Xinje XDPPro project, PLC1: XDH-60T4 (software 3.7.18 2024-11-27)

PROGRAM 梯形图

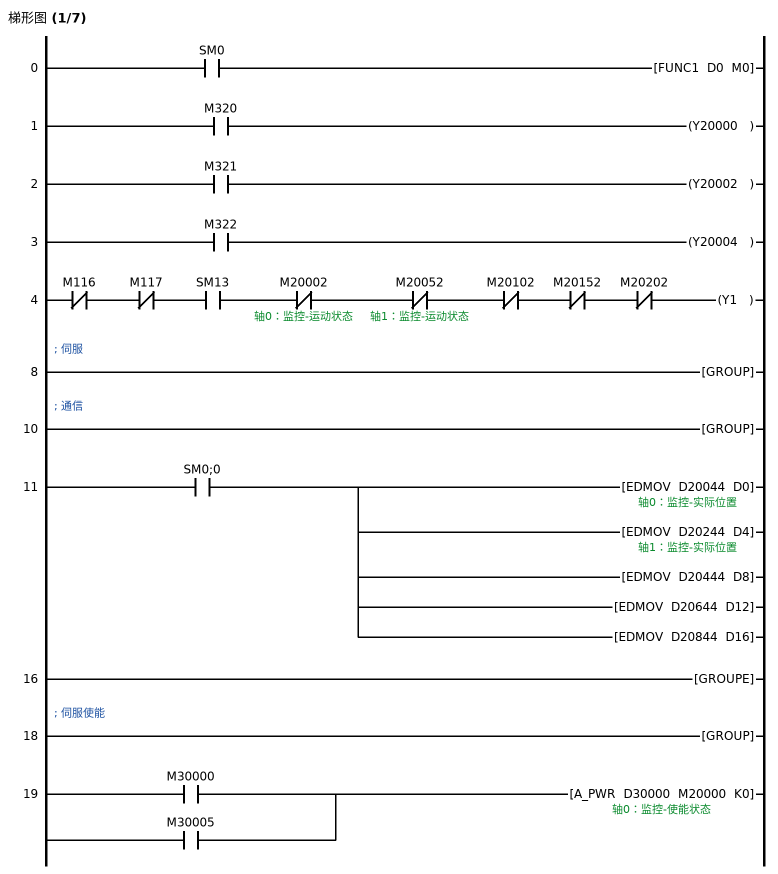
LD     SM0
FUNC1  D0 M0
LD     M320
OUT    Y20000
LD     M321
OUT    Y20002
LD     M322
OUT    Y20004
LDI    M116
ANI    M117
AND    SM13
ANI    M20002	; 轴0：监控-运动状态
ANI    M20052	; 轴1：监控-运动状态
ANI    M20102
ANI    M20152
ANI    M20202
OUT    Y1
; 伺服
GROUP
; 通信
GROUP
LD     SM0;0
EDMOV  D20044 D0	; 轴0：监控-实际位置
EDMOV  D20244 D4	; 轴1：监控-实际位置
EDMOV  D20444 D8
EDMOV  D20644 D12
EDMOV  D20844 D16
GROUPE
; 伺服使能
GROUP
LD     M30000
OR     M30005
A_PWR  D30000 M20000 K0	; 轴0：监控-使能状态

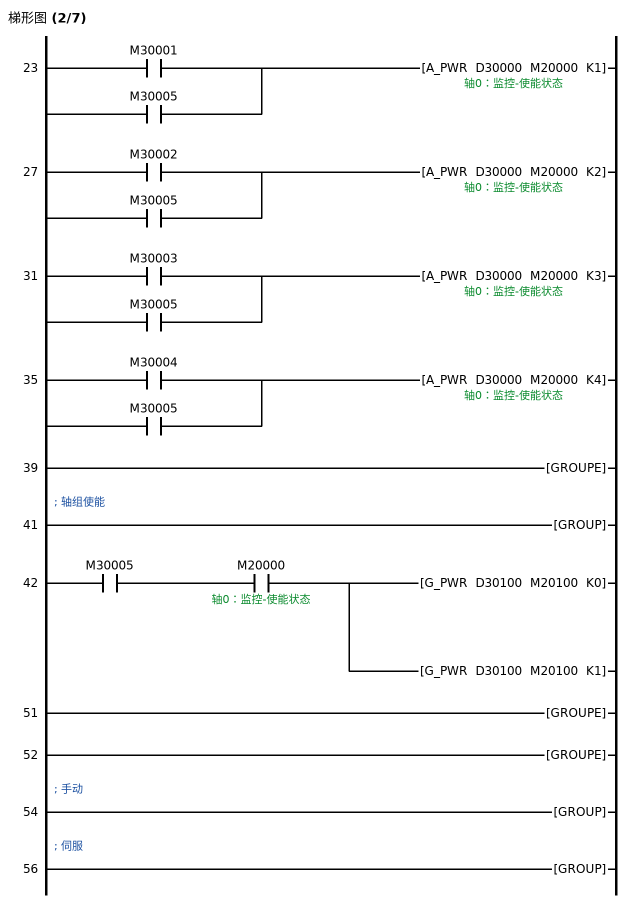
LD     M30001
OR     M30005
A_PWR  D30000 M20000 K1	; 轴0：监控-使能状态
LD     M30002
OR     M30005
A_PWR  D30000 M20000 K2	; 轴0：监控-使能状态
LD     M30003
OR     M30005
A_PWR  D30000 M20000 K3	; 轴0：监控-使能状态
LD     M30004
OR     M30005
A_PWR  D30000 M20000 K4	; 轴0：监控-使能状态
GROUPE
; 轴组使能
GROUP
LD     M30005
AND    M20000	; 轴0：监控-使能状态
G_PWR  D30100 M20100 K0
G_PWR  D30100 M20100 K1
GROUPE
GROUPE
; 手动
GROUP
; 伺服
GROUP

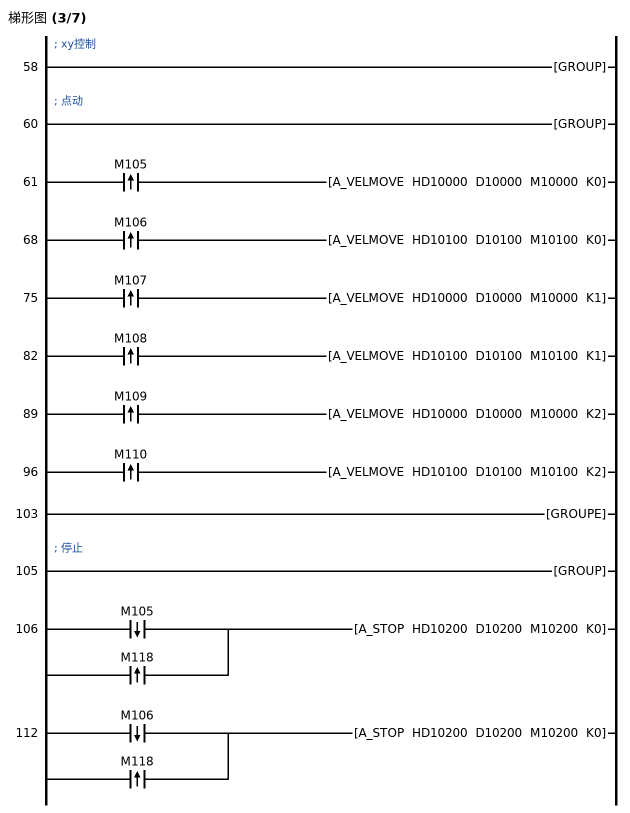
; xy控制
GROUP
; 点动
GROUP
LDP    M105
A_VELMOVE HD10000 D10000 M10000 K0
LDP    M106
A_VELMOVE HD10100 D10100 M10100 K0
LDP    M107
A_VELMOVE HD10000 D10000 M10000 K1
LDP    M108
A_VELMOVE HD10100 D10100 M10100 K1
LDP    M109
A_VELMOVE HD10000 D10000 M10000 K2
LDP    M110
A_VELMOVE HD10100 D10100 M10100 K2
GROUPE
; 停止
GROUP
LDF    M105
ORP    M118
A_STOP HD10200 D10200 M10200 K0
LDF    M106
ORP    M118
A_STOP HD10200 D10200 M10200 K0

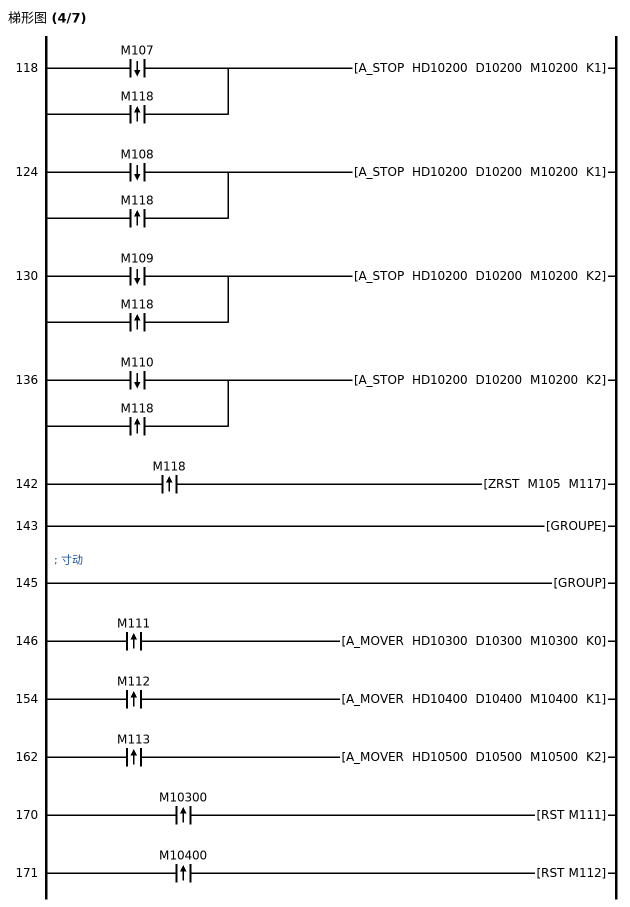
LDF    M107
ORP    M118
A_STOP HD10200 D10200 M10200 K1
LDF    M108
ORP    M118
A_STOP HD10200 D10200 M10200 K1
LDF    M109
ORP    M118
A_STOP HD10200 D10200 M10200 K2
LDF    M110
ORP    M118
A_STOP HD10200 D10200 M10200 K2
LDP    M118
ZRST   M105 M117
GROUPE
; 寸动
GROUP
LDP    M111
A_MOVER HD10300 D10300 M10300 K0
LDP    M112
A_MOVER HD10400 D10400 M10400 K1
LDP    M113
A_MOVER HD10500 D10500 M10500 K2
LDP    M10300
RST    M111
LDP    M10400
RST    M112

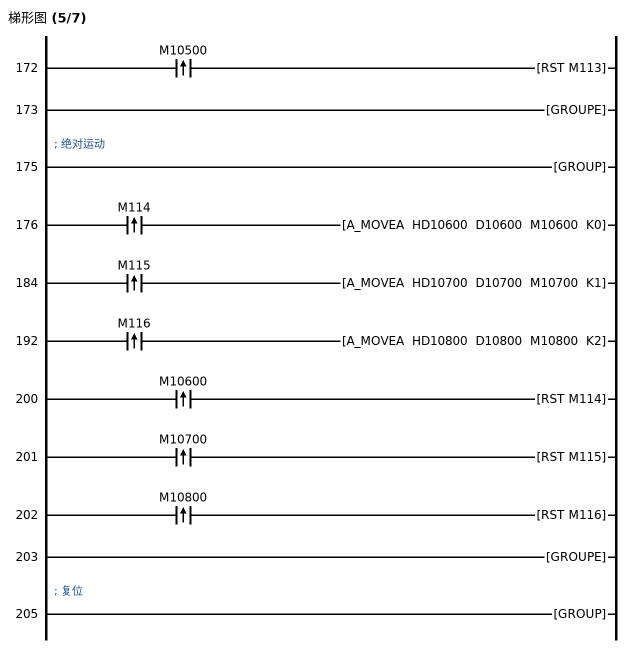
LDP    M10500
RST    M113
GROUPE
; 绝对运动
GROUP
LDP    M114
A_MOVEA HD10600 D10600 M10600 K0
LDP    M115
A_MOVEA HD10700 D10700 M10700 K1
LDP    M116
A_MOVEA HD10800 D10800 M10800 K2
LDP    M10600
RST    M114
LDP    M10700
RST    M115
LDP    M10800
RST    M116
GROUPE
; 复位
GROUP

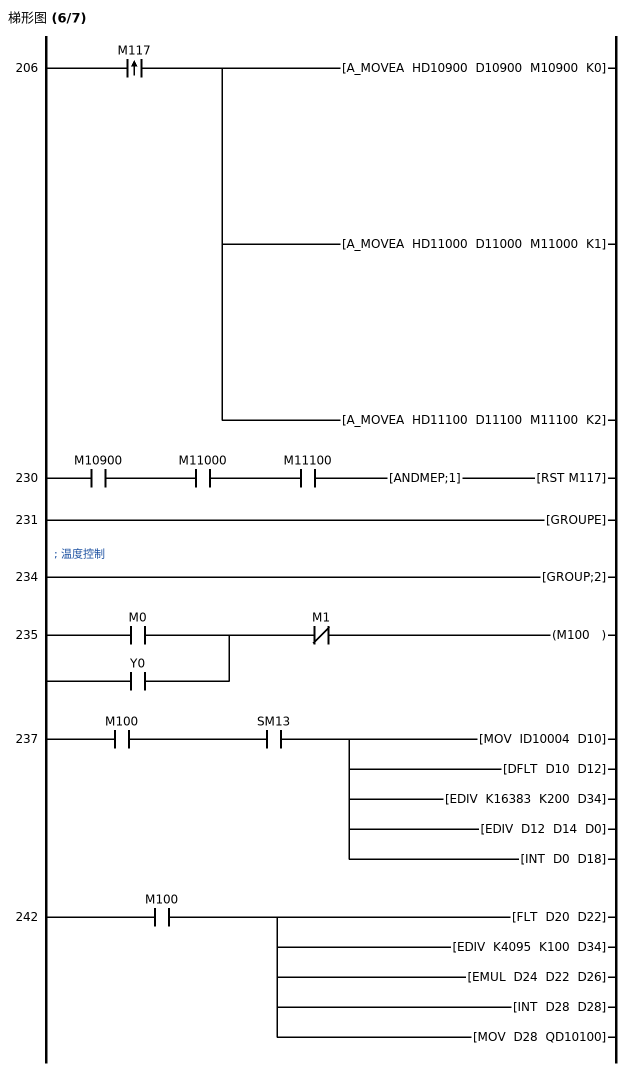
LDP    M117
A_MOVEA HD10900 D10900 M10900 K0
A_MOVEA HD11000 D11000 M11000 K1
A_MOVEA HD11100 D11100 M11100 K2
LD     M10900
AND    M11000
AND    M11100
ANDMEP;1
RST    M117
GROUPE
; 温度控制
GROUP;2
LD     M0
OR     Y0
ANI    M1
OUT    M100
LD     M100
AND    SM13
MOV    ID10004 D10
DFLT   D10 D12
EDIV   K16383 K200 D34
EDIV   D12 D14 D0
INT    D0 D18
LD     M100
FLT    D20 D22
EDIV   K4095 K100 D34
EMUL   D24 D22 D26
INT    D28 D28
MOV    D28 QD10100

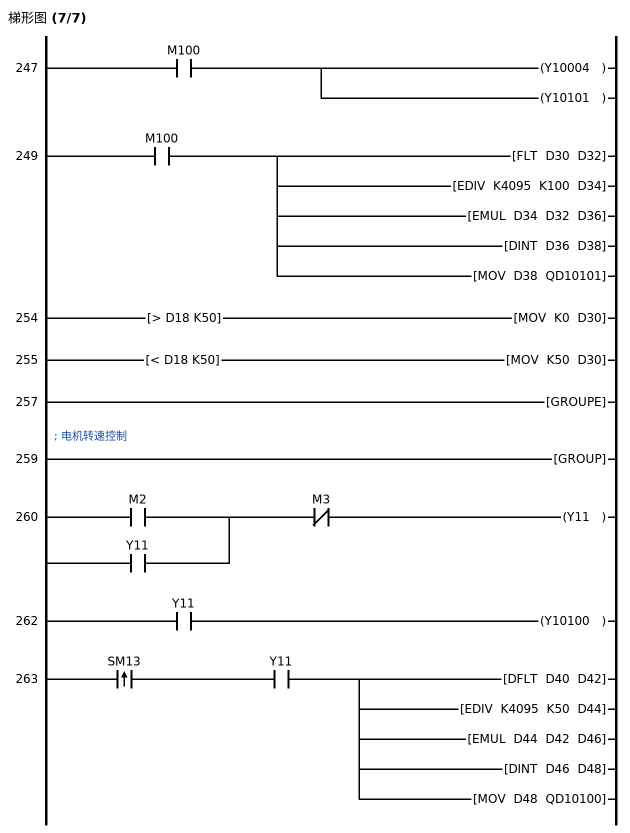
LD     M100
OUT    Y10004
OUT    Y10101
LD     M100
FLT    D30 D32
EDIV   K4095 K100 D34
EMUL   D34 D32 D36
DINT   D36 D38
MOV    D38 QD10101
LD>    D18 K50
MOV    K0 D30
LD<    D18 K50
MOV    K50 D30
GROUPE
; 电机转速控制
GROUP
LD     M2
OR     Y11
ANI    M3
OUT    Y11
LD     Y11
OUT    Y10100
LDP    SM13
AND    Y11
DFLT   D40 D42
EDIV   K4095 K50 D44
EMUL   D44 D42 D46
DINT   D46 D48
MOV    D48 QD10100

COMMENTS (devices not used above)
D20000	轴0：监控-状态机
D20200	轴1：监控-状态机
D20001	轴0：监控-错误码
D20201	轴1：监控-错误码
D20002	轴0：监控-调试模式
D20202	轴1：监控-调试模式
D20012	轴0：监控-目标位置
D20212	轴1：监控-目标位置
D20016	轴0：监控-指令位置
D20216	轴1：监控-指令位置
D20020	轴0：监控-指令速度
D20220	轴1：监控-指令速度
D20048	轴0：监控-实际速度
D20248	轴1：监控-实际速度
D20024	轴0：监控-实际加速度
D20224	轴1：监控-实际加速度
D20032	轴0：监控-指令转矩
D20232	轴1：监控-指令转矩
D20052	轴0：监控-实际转矩
D20252	轴1：监控-实际转矩
M20050	轴1：监控-使能状态
M20001	轴0：监控-错误状态
M20051	轴1：监控-错误状态
M20003	轴0：监控-定位状态
M20053	轴1：监控-定位状态
M20004	轴0：监控-原点开关
M20054	轴1：监控-原点开关
M20008	轴0：监控-指令完成状态
M20058	轴1：监控-指令完成状态
M20031	轴0：监控-正软限位
M20081	轴1：监控-正软限位
M20032	轴0：监控-负软限位
M20082	轴1：监控-负软限位
M20029	轴0：监控-正硬限位
M20079	轴1：监控-正硬限位
M20030	轴0：监控-负硬限位
M20080	轴1：监控-负硬限位
D20104	轴0：调试-启用轴调试
D20304	轴1：调试-启用轴调试
D20105	轴0：调试-运动类型
D20305	轴1：调试-运动类型
D20108	轴0：调试-目标位置
D20308	轴1：调试-目标位置
D20112	轴0：调试-速度
D20312	轴1：调试-速度
D20116	轴0：调试-加速度
D20316	轴1：调试-加速度
D20120	轴0：调试-减速度
D20320	轴1：调试-减速度
D20124	轴0：调试-加加速度
D20324	轴1：调试-加加速度
D20128	轴0：调试-修改位置值
D20328	轴1：调试-修改位置值
D20132	轴0：调试-原点偏移
D20332	轴1：调试-原点偏移
D20136	轴0：调试-转矩给定
D20336	轴1：调试-转矩给定
D20140	轴0：调试-速度限制
D20340	轴1：调试-速度限制
D20144	轴0：调试-转矩斜坡
D20344	轴1：调试-转矩斜坡
M20020	轴0：调试-使能
M20070	轴1：调试-使能
M20022	轴0：调试-目标位置运动
M20072	轴1：调试-目标位置运动
M20023	轴0：调试-正向点动
M20073	轴1：调试-正向点动
M20024	轴0：调试-反向点动
M20074	轴1：调试-反向点动
M20025	轴0：调试-回原点
M20075	轴1：调试-回原点
M20026	轴0：调试-复位
M20076	轴1：调试-复位
M20028	轴0：调试-修改位置
M20078	轴1：调试-修改位置

C FUNCTION BLOCK func1.fcb
/* #EXPORT_ENTRY_BEGIN(FUNC1)
//    类型              模式             个数               映射          注释
W = { type = "PINT16S", mode = [In,Out], count = "unknown", map = [D,HD], comment = "" }
B = { type = "PBIT"   , mode = [In,Out], count = "unknown", map = [M,HM], comment = "" }
#EXPORT_ENTRY_END */
/*************************************************************************
 * FunctionBlockName:  FUNC1
 * Version:            1.0.0
 * Author:
 * UpdateTime:         2025-05-08 19:20:47
 * Comment:
**************************************************************************/

/**
 * @summary
 * @param W
 * @param B
 */
void FUNC1 ( PINT16S W, PBIT B )
{
#define SysRegAddr_HD_D_HM_M
#include "func1.h"
//参数赋值
    FDHD[10004] = FDHD[10000] * 10;
    FDHD[10008] = FDHD[10000] * 10;
    FDHD[10012] = FDHD[10000] * 100;

    FDHD[10100] = FDHD[10000] * -1;

    FDHD[10104] = FDHD[10000] * 10;
    FDHD[10108] = FDHD[10000] * 10;
    FDHD[10112] = FDHD[10000] * 100;

    FDHD[10200] = FDHD[10000] * 10;
    FDHD[10204] = FDHD[10000] * 100;

    FDHD[10304] = FDHD[10000];
    FDHD[10404] = FDHD[10000];
    FDHD[10504] = FDHD[10000];

    FDHD[10308] = FDHD[10000] * 10;
    FDHD[10408] = FDHD[10000] * 10;
    FDHD[10508] = FDHD[10000] * 10;

    FDHD[10312] = FDHD[10000] * 10;
    FDHD[10412] = FDHD[10000] * 10;
    FDHD[10512] = FDHD[10000] * 10;

    FDHD[10316] = FDHD[10000] * 100;
    FDHD[10416] = FDHD[10000] * 100;
    FDHD[10516] = FDHD[10000] * 100;

    FDHD[10604] = FDHD[10000];
    FDHD[10704] = FDHD[10000];
    FDHD[10804] = FDHD[10000];

    FDHD[10608] = FDHD[10000] * 10;
    FDHD[10708] = FDHD[10000] * 10;
    FDHD[10808] = FDHD[10000] * 10;

    FDHD[10612] = FDHD[10000] * 10;
    FDHD[10712] = FDHD[10000] * 10;
    FDHD[10812] = FDHD[10000] * 10;

    FDHD[10616] = FDHD[10000] * 100;
    FDHD[10716] = FDHD[10000] * 100;
    FDHD[10816] = FDHD[10000] * 100;

    FDHD[10900] = 0;
    FDHD[11000] = 0;
    FDHD[11100] = 0;

    FDHD[10904] = FDHD[10000];
    FDHD[11004] = FDHD[10000];
    FDHD[11104] = FDHD[10000];

    FDHD[10908] = FDHD[10000] * 10;
    FDHD[11008] = FDHD[10000] * 10;
    FDHD[11108] = FDHD[10000] * 10;

    FDHD[10912] = FDHD[10000] * 10;
    FDHD[11012] = FDHD[10000] * 10;
    FDHD[11112] = FDHD[10000] * 10;

    FDHD[10916] = FDHD[10000] * 100;
    FDHD[11016] = FDHD[10000] * 100;
    FDHD[11116] = FDHD[10000] * 100;

    FDHD[12004] = FDHD[12000] * 10;
    FDHD[12008] = FDHD[12000] * 10;
    FDHD[12012] = FDHD[12000] * 100;

    FDHD[12100] = FDHD[12000] * -1;

    FDHD[12104] = FDHD[12000] * 10;
    FDHD[12108] = FDHD[12000] * 10;
    FDHD[12112] = FDHD[12000] * 100;

    FDHD[10200] = FDHD[12000] * 10;
    FDHD[12204] = FDHD[12000] * 100;

    FDHD[12304] = FDHD[12000];
    FDHD[12404] = FDHD[12000];

    FDHD[12308] = FDHD[12000] * 10;
    FDHD[12408] = FDHD[12000] * 10;

    FDHD[12312] = FDHD[12000] * 10;
    FDHD[12412] = FDHD[12000] * 10;

    FDHD[12316] = FDHD[12000] * 100;
    FDHD[12416] = FDHD[12000] * 100;

    FDHD[12504] = FDHD[12000];
    FDHD[12604] = FDHD[12000];

    FDHD[12508] = FDHD[12000] * 10;
    FDHD[12608] = FDHD[12000] * 10;

    FDHD[12512] = FDHD[12000] * 10;
    FDHD[12612] = FDHD[12000] * 10;

    FDHD[12516] = FDHD[12000] * 100;
    FDHD[12616] = FDHD[12000] * 100;

    FDHD[12704] = FDHD[12000];

    FDHD[12708] = FDHD[12000] * 10;

    FDHD[12712] = FDHD[12000] * 10;

    FDHD[12716] = FDHD[12000] * 100;

    D[13100] = 200 * D[102];
    D[13104] = 800 * D[103];
    D[13108] = 0;


//自动参数赋值
    switch ( D[100] )
    {
    case 1://取物点
        D[13100] = 200;
        D[13104] = 800;
        D[13108] = 0;
        break;
    case 2://z下降
        D[13100] = 200;
        D[13104] = 800;
        D[13108] = -450;
        break;
    case 4://z上升
        D[13100] = 200;
        D[13104] = 800;
        D[13108] = 0;
        break;
    case 5://前往码垛点

        switch ( D[101] )
        {
        case 1:
            D[13100] = 200;
            D[13104] = -200;
            break;
        case 2:
            D[13100] = 400;
            D[13104] = -200;
            break;
        case 3:
            D[13100] = 200;
            D[13104] = 0;
            break;
        case 4:
            D[13100] = 400;
            D[13104] = 0;
            break;

        }
    case 6://z下降
        D[13108] = -300;
        break;

    case 7://z上升
        D[13108] = 0;
        break;

    case 8://复位
        D[13100] = 0;
        D[13104] = 0;
        D[13108] = 0;
        break;


    }
    
    switch(D[102])
    {
    	case 2: 
        D[13300] = 0;
        D[13304] = 0;
    	break;
    	case 4:
    	D[13300] = 0;
        D[13304] = 400;
        break;
    }
}

C FILE func1.h
#ifndef	_HDY_H
#define	_HDY_H

    /*****sky**********sky**********sky**********sky**********sky*****
    W[0]    系统默认的调用单字整型
    DW[0]   系统默认的调用双字整型
    FW[0]   系统默认的调用浮点型
    *****sky**********sky**********sky**********sky**********sky*****/
    #define 	DD      *(INT32S*)&D    //举例：DD[0]=1;   将D[0]-D[1]作为双字整数，对其赋值为1；    注意[]中必须是非负偶数
    #define 	FDD     *(FP32*)&D      //举例：FDD[0]=1;  将D[0]-D[1]作为单精度浮点数，对其赋值为1；注意[]中必须是非负偶数
 	#define 	DFD     *(FP64*)&D      //举例：DFD[0]=1;  将D[0]-D[3]作为双精度浮点数，对其赋值为1；注意[]中必须是非负偶数，且是4的整倍数
 	#define     UD      *(long long*)&D //举例：UD[0]=1;   将D[0]-D[3]作为四字整数，对其赋值为1；    注意[]中必须是非负偶数，且是4的整倍数
 	#define 	DHD     *(INT32S*)&HD   //举例：DHD[0]=1;  将HD[0]-HD[1]作为双字数，对其赋值为1；      注意[]中必须是非负偶数
 	#define 	FHD     *(FP32*)&HD     //举例：FHD[0]=1;  将HD[0]-HD[1]作为单精度浮点数，对其赋值为1；注意[]中必须是非负偶数
 	#define 	FDHD    *(FP64*)&HD     //举例：FDHD[0]=1; 将HD[0]-HD[3]作为双精度浮点数，对其赋值为1；注意[]中必须是非负偶数，且是4的整倍数
 	#define 	UHD     *(long long*)&HD//举例：UHD[0]=1;  将HD[0]-HD[3]作为四字整数，对其赋值为1；    注意[]中必须是非负偶数，且是4的整倍数

#endif